TYPE CM_Sensor_WRN :
STRUCT
END_STRUCT
END_TYPE

(* stored: Version 1.1.0.1, ProductVersion 3.1.4024.12
   DUT CM_Sensor_WRN: Id {a8252369-732c-4714-89e4-4e7fc7eb704e} *)
